TYPE InputBase_8311D824 :
STRUCT
END_STRUCT
END_TYPE

(* stored: Version 1.2.0.0, ProductVersion 3.1.4024.11
   DUT InputBase_8311D824: Id {68401f04-7ebd-42c0-a25e-8e0662111e15} *)
